	(*═════════════════════════════════════════════════════════*)
	(*  Communication and PLC    *)
	(*═════════════════════════════════════════════════════════*)
	PLC_r_CPUload                                              , (* REAL *)
	PLC_e_ProfinetState                                        , (* eNetcomState *)
	PLC_e_EthercatState                                        , (* eNetcomState *)
	Cooling_CoolingSystemMode                                  , (* eCoolingSystemState *)
	Cooling_HeatPumpStatus                                     , (* eHeatPumpState *)
	Cooling_r_CoolantTemperature                               , (* REAL *)
	Cooling_r_CoolantPressure                                  , (* REAL *)
	Cooling_r_EnclosureDewpoint                                , (* REAL *)
	Cooling_ui_DehumRemainingTime                              , (* UINT *)
	Cooling_HeatPumpSystem_HeatPumpStatus                      , (* eHeatPumpState *)
	Cooling_HeatPumpSystem_PrimaryHeatpumpGet_HeatPumpState    , (* eHeatPumpState *)
	Cooling_HeatPumpSystem_PrimaryHeatpumpGet_Setpoint         , (* REAL *)
	Cooling_HeatPumpSystem_PrimaryHeatpumpGet_Events_b_CommWarning, (* BOOL *)
	Cooling_HeatPumpSystem_PrimaryHeatpumpGet_Events_b_ProbeError, (* BOOL *)
	Cooling_HeatPumpSystem_PrimaryHeatpumpGet_Events_b_PressureError, (* BOOL *)
	Cooling_HeatPumpSystem_PrimaryHeatpumpGet_Events_b_CompressorError, (* BOOL *)
	Cooling_HeatPumpSystem_PrimaryHeatpumpGet_Events_b_ValveError, (* BOOL *)
	Cooling_HeatPumpSystem_PrimaryHeatpumpGet_Events_b_FanError, (* BOOL *)
	Cooling_HeatPumpSystem_PrimaryHeatpumpGet_Events_b_PumpError, (* BOOL *)
	Cooling_HeatPumpSystem_PrimaryHeatpumpGet_Events_b_WaterTempError, (* BOOL *)
	Cooling_HeatPumpSystem_PrimaryHeatpumpGet_Events_b_IOError , (* BOOL *)
	Cooling_HeatPumpSystem_PrimaryHeatpumpGet_Events_b_HeatpumpPreheatingActive, (* BOOL *)
	Cooling_HeatPumpSystem_PrimaryHeatpumpGet_Events_b_TooColdForHeatpumpHeating, (* BOOL *)
	Cooling_HeatPumpSystem_PrimaryHeatpumpGet_HeatpumpData_i_FW_Version, (* INT *)
	Cooling_HeatPumpSystem_PrimaryHeatpumpGet_HeatpumpData_i_FW_release, (* INT *)
	Cooling_HeatPumpSystem_PrimaryHeatpumpGet_HeatpumpData_w_FW_Subrelease, (* WORD *)
	Cooling_HeatPumpSystem_PrimaryHeatpumpGet_HeatpumpData_w_FW_creationDate, (* WORD *)
	Cooling_HeatPumpSystem_PrimaryHeatpumpGet_HeatpumpData_w_Serialnumber_0  , (* WORD *)
	Cooling_HeatPumpSystem_PrimaryHeatpumpGet_HeatpumpData_w_Serialnumber_1  , (* WORD *)
	Cooling_HeatPumpSystem_PrimaryHeatpumpGet_HeatpumpData_w_Serialnumber_2  , (* WORD *)
	Cooling_HeatPumpSystem_PrimaryHeatpumpGet_HeatpumpData_w_Serialnumber_3  , (* WORD *)
	Cooling_HeatPumpSystem_PrimaryHeatpumpGet_HeatpumpData_w_Serialnumber_4  , (* WORD *)
	Cooling_HeatPumpSystem_PrimaryHeatpumpGet_HeatpumpData_w_Serialnumber_5  , (* WORD *)
	Cooling_HeatPumpSystem_PrimaryHeatpumpGet_HeatpumpData_w_Serialnumber_6  , (* WORD *)
	Cooling_HeatPumpSystem_PrimaryHeatpumpGet_HeatpumpData_w_Serialnumber_7  , (* WORD *)
	Cooling_HeatPumpSystem_PrimaryHeatpumpGet_HeatpumpData_w_Serialnumber_8  , (* WORD *)
	Cooling_HeatPumpSystem_PrimaryHeatpumpGet_HeatpumpData_w_Serialnumber_9  , (* WORD *)
	Cooling_HeatPumpSystem_PrimaryHeatpumpGet_HeatpumpData_w_Serialnumber_10 , (* WORD *)
	Cooling_HeatPumpSystem_PrimaryHeatpumpGet_HeatpumpData_w_Serialnumber_11 , (* WORD *)
	Cooling_HeatPumpSystem_PrimaryHeatpumpGet_HeatpumpData_w_Serialnumber_12 , (* WORD *)
	Cooling_HeatPumpSystem_PrimaryHeatpumpGet_HeatpumpData_w_Serialnumber_13 , (* WORD *)
	Cooling_HeatPumpSystem_PrimaryHeatpumpGet_HeatpumpData_w_Serialnumber_14 , (* WORD *)
	Cooling_HeatPumpSystem_PrimaryHeatpumpGet_HeatpumpData_w_Serialnumber_15 , (* WORD *)
	Cooling_HeatPumpSystem_PrimaryHeatpumpGet_HeatpumpData_w_Serialnumber_16 , (* WORD *)
	Cooling_HeatPumpSystem_PrimaryHeatpumpGet_HeatpumpData_w_Serialnumber_17 , (* WORD *)
	Cooling_HeatPumpSystem_PrimaryHeatpumpGet_HeatpumpData_i_OperatingHours, (* INT *)
	Cooling_HeatPumpSystem_PrimaryHeatpumpGet_HeatpumpData_r_CoolantPower, (* REAL *)
	Cooling_HeatPumpSystem_PrimaryHeatpumpGet_HeatpumpData_r_InletWaterTemp, (* REAL *)
	Cooling_HeatPumpSystem_PrimaryHeatpumpGet_HeatpumpData_r_OutletWaterTemp, (* REAL *)
	Cooling_HeatPumpSystem_PrimaryHeatpumpGet_HeatpumpData_r_HighPressure, (* REAL *)
	Cooling_HeatPumpSystem_PrimaryHeatpumpGet_HeatpumpData_r_LowPressure, (* REAL *)
	Cooling_HeatPumpSystem_PrimaryHeatpumpGet_HeatpumpData_r_CompInputTemp, (* REAL *)
	Cooling_HeatPumpSystem_PrimaryHeatpumpGet_HeatpumpData_r_OutdoorTemp, (* REAL *)
	Cooling_HeatPumpSystem_PrimaryHeatpumpGet_HeatpumpData_r_CompOutputTemp, (* REAL *)
	Cooling_HeatPumpSystem_PrimaryHeatpumpGet_HeatpumpData_ui_WaterFlowRate, (* UINT *)
	Cooling_HeatPumpSystem_PrimaryHeatpumpGet_HeatpumpData_w_ErrorList_1  , (* WORD *)
	Cooling_HeatPumpSystem_PrimaryHeatpumpGet_HeatpumpData_w_ErrorList_2  , (* WORD *)
	Cooling_HeatPumpSystem_PrimaryHeatpumpGet_HeatpumpData_w_ErrorList_3  , (* WORD *)
	Cooling_HeatPumpSystem_PrimaryHeatpumpGet_HeatpumpData_w_ErrorList_4  , (* WORD *)
	Cooling_HeatPumpSystem_PrimaryHeatpumpGet_HeatpumpData_w_ErrorList_5  , (* WORD *)
	Cooling_HeatPumpSystem_PrimaryHeatpumpGet_HeatpumpData_w_ErrorList_6  , (* WORD *)
	Cooling_HeatPumpSystem_PrimaryHeatpumpGet_HeatpumpData_w_ErrorList_7  , (* WORD *)
	Cooling_HeatPumpSystem_PrimaryHeatpumpGet_HeatpumpData_r_FanSpeedPCT, (* REAL *)
	Cooling_HeatPumpSystem_PrimaryHeatpumpGet_HeatpumpData_r_PumpSpeedPCT, (* REAL *)
	Cooling_HeatPumpSystem_PrimaryHeatpumpGet_HeatpumpData_r_SetpointHeating, (* REAL *)
	Cooling_HeatPumpSystem_PrimaryHeatpumpGet_HeatpumpData_r_SetpointCooling, (* REAL *)
	Cooling_HeatPumpSystem_PrimaryHeatpumpGet_HeatpumpData_b_DefrostingActive, (* BOOL *)
	Cooling_HeatPumpSystem_SecondaryHeatpumpGet_HeatPumpState  , (* eHeatPumpState *)
	Cooling_HeatPumpSystem_SecondaryHeatpumpGet_Setpoint       , (* REAL *)
	Cooling_HeatPumpSystem_SecondaryHeatpumpGet_Events_b_CommWarning, (* BOOL *)
	Cooling_HeatPumpSystem_SecondaryHeatpumpGet_Events_b_ProbeError, (* BOOL *)
	Cooling_HeatPumpSystem_SecondaryHeatpumpGet_Events_b_PressureError, (* BOOL *)
	Cooling_HeatPumpSystem_SecondaryHeatpumpGet_Events_b_CompressorError, (* BOOL *)
	Cooling_HeatPumpSystem_SecondaryHeatpumpGet_Events_b_ValveError, (* BOOL *)
	Cooling_HeatPumpSystem_SecondaryHeatpumpGet_Events_b_FanError, (* BOOL *)
	Cooling_HeatPumpSystem_SecondaryHeatpumpGet_Events_b_PumpError, (* BOOL *)
	Cooling_HeatPumpSystem_SecondaryHeatpumpGet_Events_b_WaterTempError, (* BOOL *)
	Cooling_HeatPumpSystem_SecondaryHeatpumpGet_Events_b_IOError, (* BOOL *)
	Cooling_HeatPumpSystem_SecondaryHeatpumpGet_Events_b_HeatpumpPreheatingActive, (* BOOL *)
	Cooling_HeatPumpSystem_SecondaryHeatpumpGet_Events_b_TooColdForHeatpumpHeating, (* BOOL *)
	Cooling_HeatPumpSystem_SecondaryHeatpumpGet_HeatpumpData_i_FW_Version, (* INT *)
	Cooling_HeatPumpSystem_SecondaryHeatpumpGet_HeatpumpData_i_FW_release, (* INT *)
	Cooling_HeatPumpSystem_SecondaryHeatpumpGet_HeatpumpData_w_FW_Subrelease, (* WORD *)
	Cooling_HeatPumpSystem_SecondaryHeatpumpGet_HeatpumpData_w_FW_creationDate, (* WORD *)
	Cooling_HeatPumpSystem_SecondaryHeatpumpGet_HeatpumpData_w_Serialnumber_0  , (* WORD *)
	Cooling_HeatPumpSystem_SecondaryHeatpumpGet_HeatpumpData_w_Serialnumber_1  , (* WORD *)
	Cooling_HeatPumpSystem_SecondaryHeatpumpGet_HeatpumpData_w_Serialnumber_2  , (* WORD *)
	Cooling_HeatPumpSystem_SecondaryHeatpumpGet_HeatpumpData_w_Serialnumber_3  , (* WORD *)
	Cooling_HeatPumpSystem_SecondaryHeatpumpGet_HeatpumpData_w_Serialnumber_4  , (* WORD *)
	Cooling_HeatPumpSystem_SecondaryHeatpumpGet_HeatpumpData_w_Serialnumber_5  , (* WORD *)
	Cooling_HeatPumpSystem_SecondaryHeatpumpGet_HeatpumpData_w_Serialnumber_6  , (* WORD *)
	Cooling_HeatPumpSystem_SecondaryHeatpumpGet_HeatpumpData_w_Serialnumber_7  , (* WORD *)
	Cooling_HeatPumpSystem_SecondaryHeatpumpGet_HeatpumpData_w_Serialnumber_8  , (* WORD *)
	Cooling_HeatPumpSystem_SecondaryHeatpumpGet_HeatpumpData_w_Serialnumber_9  , (* WORD *)
	Cooling_HeatPumpSystem_SecondaryHeatpumpGet_HeatpumpData_w_Serialnumber_10 , (* WORD *)
	Cooling_HeatPumpSystem_SecondaryHeatpumpGet_HeatpumpData_w_Serialnumber_11 , (* WORD *)
	Cooling_HeatPumpSystem_SecondaryHeatpumpGet_HeatpumpData_w_Serialnumber_12 , (* WORD *)
	Cooling_HeatPumpSystem_SecondaryHeatpumpGet_HeatpumpData_w_Serialnumber_13 , (* WORD *)
	Cooling_HeatPumpSystem_SecondaryHeatpumpGet_HeatpumpData_w_Serialnumber_14 , (* WORD *)
	Cooling_HeatPumpSystem_SecondaryHeatpumpGet_HeatpumpData_w_Serialnumber_15 , (* WORD *)
	Cooling_HeatPumpSystem_SecondaryHeatpumpGet_HeatpumpData_w_Serialnumber_16 , (* WORD *)
	Cooling_HeatPumpSystem_SecondaryHeatpumpGet_HeatpumpData_w_Serialnumber_17 , (* WORD *)
	Cooling_HeatPumpSystem_SecondaryHeatpumpGet_HeatpumpData_i_OperatingHours, (* INT *)
	Cooling_HeatPumpSystem_SecondaryHeatpumpGet_HeatpumpData_r_CoolantPower, (* REAL *)
	Cooling_HeatPumpSystem_SecondaryHeatpumpGet_HeatpumpData_r_InletWaterTemp, (* REAL *)
	Cooling_HeatPumpSystem_SecondaryHeatpumpGet_HeatpumpData_r_OutletWaterTemp, (* REAL *)
	Cooling_HeatPumpSystem_SecondaryHeatpumpGet_HeatpumpData_r_HighPressure, (* REAL *)
	Cooling_HeatPumpSystem_SecondaryHeatpumpGet_HeatpumpData_r_LowPressure, (* REAL *)
	Cooling_HeatPumpSystem_SecondaryHeatpumpGet_HeatpumpData_r_CompInputTemp, (* REAL *)
	Cooling_HeatPumpSystem_SecondaryHeatpumpGet_HeatpumpData_r_OutdoorTemp, (* REAL *)
	Cooling_HeatPumpSystem_SecondaryHeatpumpGet_HeatpumpData_r_CompOutputTemp, (* REAL *)
	Cooling_HeatPumpSystem_SecondaryHeatpumpGet_HeatpumpData_ui_WaterFlowRate, (* UINT *)
	Cooling_HeatPumpSystem_SecondaryHeatpumpGet_HeatpumpData_w_ErrorList_1  , (* WORD *)
	Cooling_HeatPumpSystem_SecondaryHeatpumpGet_HeatpumpData_w_ErrorList_2  , (* WORD *)
	Cooling_HeatPumpSystem_SecondaryHeatpumpGet_HeatpumpData_w_ErrorList_3  , (* WORD *)
	Cooling_HeatPumpSystem_SecondaryHeatpumpGet_HeatpumpData_w_ErrorList_4  , (* WORD *)
	Cooling_HeatPumpSystem_SecondaryHeatpumpGet_HeatpumpData_w_ErrorList_5  , (* WORD *)
	Cooling_HeatPumpSystem_SecondaryHeatpumpGet_HeatpumpData_w_ErrorList_6  , (* WORD *)
	Cooling_HeatPumpSystem_SecondaryHeatpumpGet_HeatpumpData_w_ErrorList_7  , (* WORD *)
	Cooling_HeatPumpSystem_SecondaryHeatpumpGet_HeatpumpData_r_FanSpeedPCT, (* REAL *)
	Cooling_HeatPumpSystem_SecondaryHeatpumpGet_HeatpumpData_r_PumpSpeedPCT, (* REAL *)
	Cooling_HeatPumpSystem_SecondaryHeatpumpGet_HeatpumpData_r_SetpointHeating, (* REAL *)
	Cooling_HeatPumpSystem_SecondaryHeatpumpGet_HeatpumpData_r_SetpointCooling, (* REAL *)
	Cooling_HeatPumpSystem_SecondaryHeatpumpGet_HeatpumpData_b_DefrostingActive, (* BOOL *)
	Cooling_Events_b_SystemOvertemperatureWarning              , (* BOOL *)
	Cooling_Events_b_SystemUnderTemperatureWarning             , (* BOOL *)
	Cooling_Events_b_CoolingSystemFuseFailure                  , (* BOOL *)
	Cooling_Events_b_ACwaterPumpTimeOut                        , (* BOOL *)
	Cooling_Events_b_InverterLoopValveStuck                    , (* BOOL *)
	Cooling_Events_b_BattLoopValveStuck                        , (* BOOL *)
	Cooling_Events_b_FancoilLoopValveStuck                     , (* BOOL *)
	Cooling_Events_b_DCpumpPressureFault                       , (* BOOL *)
	Cooling_Events_b_DCpumpTimeout                             , (* BOOL *)
	Cooling_Events_b_CoolingLoopIdlePressureWarning            , (* BOOL *)
	Cooling_Events_b_CoolingLoopIdlePressureError              , (* BOOL *)
	Cooling_Events_b_InverterCoolingLoopError                  , (* BOOL *)
	Cooling_Events_b_HeatpumpWarning                           , (* BOOL *)
	Cooling_Events_b_HeatPumpError                             , (* BOOL *)
	Cooling_Events_b_CoolantTempTooLow                         , (* BOOL *)
	Cooling_Events_b_CoolantTempLow                            , (* BOOL *)
	Cooling_Events_b_CoolantTempTooHigh                        , (* BOOL *)
	Cooling_Events_b_CoolantTempHigh                           , (* BOOL *)
	Router_Device_SystemUptime                                 , (* UDINT *)
	Router_Device_Temperature                                  , (* REAL *)
	Router_Device_RouterSerial                                 , (* STRING(32) *)
	Router_GPS_Latitude                                        , (* REAL *)
	Router_GPS_Longitude                                       , (* REAL *)
	Router_GPS_FixTime                                         , (* STRING(32) *)
	Router_GPS_DateTime                                        , (* DT *)
	Router_GPS_Speed                                           , (* REAL *)
	Router_GPS_SatCount                                        , (* UINT *)
	Router_GPS_Accuracy                                        , (* REAL *)
	Router_Mobile_NetworkOperator                              , (* STRING(32) *)
	Router_Mobile_NetworkInfo                                  , (* STRING(32) *)
	Router_Mobile_NetworkType                                  , (* STRING(32) *)
	Router_Mobile_RSSI                                         , (* DINT *)
	Router_Mobile_ui_Sim1DataSendMonth                         , (* UINT *)
	Router_Mobile_ui_Sim1DataReceivedMonth                     , (* UINT *)
	Router_Mobile_ui_Sim2DataSendMonth                         , (* UINT *)
	Router_Mobile_ui_Sim2DataReceivedMonth                     , (* UINT *)
	Router_Mobile_s_EmergencySMSNumber                         , (* STRING(20) *)
	Router_Mobile_s_SecondarySMSNumber                         , (* STRING(20) *)
	Router_Mobile_s_EmergencySMSDevName                        , (* STRING(18) *)
	Router_Mobile_st_LatestSMSMessage                          , (* STRING(80) *)
	Router_Mobile_ModemState                                   , (* eModemState *)
	Router_Mobile_NetworkState                                 , (* eNetworkState *)
	Router_Mobile_ui_ActiveSim                                 , (* UINT *)
	Router_Mobile_SimStatus                                    , (* eSimState *)
	Router_Wifi_WifiClienModeStatus                            , (* eWifiStatus *)
	Router_Wifi_WifiAPModeStatus                               , (* eWifiStatus *)
	Router_Wifi_WifiApNumberOfClients                          , (* UINT *)
	Router_e_SMSStatus                                         , (* eSMSStatus *)
	Router_Events_b_MBCommWarning                              , (* BOOL *)
	Router_Events_b_NoSimWarning                               , (* BOOL *)
	Router_Events_b_NoNetworkWarning                           , (* BOOL *)
	Router_Events_b_noGPSFixWarning                            , (* BOOL *)
	Router_Events_b_SMSNotSendError                            , (* BOOL *)
	Router_Events_b_NoSMSNumberAvailable                       , (* BOOL *)
	Router_Events_b_TimeUpdateFailed                           , (* BOOL *)

	(*═════════════════════════════════════════════════════════*)
	(*  External Systems and I/O    *)
	(*═════════════════════════════════════════════════════════*)
	controlfb_control_b_start                                  , (* BOOL *)
	controlfb_control_b_stop                                   , (* BOOL *)
	controlfb_control_b_shutdown                               , (* BOOL *)
	controlfb_control_b_Reset                                  , (* BOOL *)
	controlfb_control_b_SystemShutdown                         , (* BOOL *)
	controlfb_control_b_EMstop                                 , (* BOOL *)
	controlfb_control_b_ClearHistory                           , (* BOOL *)
	controlfb_control_b_ActivateSettings                       , (* BOOL *)
	controlfb_control_b_startDeHum                             , (* BOOL *)
	controlfb_Operation_inputgrid_b_SyncClose                  , (* BOOL *)
	controlfb_Operation_Genset_b_manualStart                   , (* BOOL *)
	controlfb_Operation_PSB_b_SyncClose                        , (* BOOL *)
	controlfb_Operation_charger_b_StartCharging                , (* BOOL *)
	controlfb_Operation_charger_b_ResetCharger                 , (* BOOL *)
	controlfb_Operation_system_r_NominalVoltage                , (* REAL *)
	controlfb_Operation_system_r_NominalFrequency              , (* REAL *)
	controlfb_Operation_system_r_Pset                          , (* REAL *)
	controlfb_Operation_system_r_Qset                          , (* REAL *)
	controlfb_Operation_system_r_PFset                         , (* REAL *)
	controlfb_Operation_system_b_PFsetEnable                   , (* BOOL *)
	controlfb_Operation_system_b_SounderMute                   , (* BOOL *)
	controlfb_Operation_system_b_SounderTest                   , (* BOOL *)
	controlfb_Operation_system_b_GenGridModeTrans              , (* BOOL *)
	controlfb_Operation_system_b_GridTakeOverEnable            , (* BOOL *)
	controlfb_Operation_parallel_b_DetectSlaves                , (* BOOL *)
	controlfb_Operation_parallel_r_ActivePowerSlave1           , (* REAL *)
	controlfb_Operation_parallel_r_ReactivePowerSlave1         , (* REAL *)
	controlfb_Operation_parallel_r_ActivePowerSlave2           , (* REAL *)
	controlfb_Operation_parallel_r_ReactivePowerSlave2         , (* REAL *)
	controlfb_Operation_BMS_b_ManualStartHVDC                  , (* BOOL *)
	controlfb_SoftSettings_inputgrid_PeakshaveMode             , (* ePeakshaveMode *)
	controlfb_SoftSettings_inputgrid_setpointTimeslot1_r_SocTarget, (* REAL *)
	controlfb_SoftSettings_inputgrid_setpointTimeslot1_r_IdleChargePower, (* REAL *)
	controlfb_SoftSettings_inputgrid_setpointTimeslot1_r_FeedInCurrentLimitSoft, (* REAL *)
	controlfb_SoftSettings_inputgrid_setpointTimeslot1_r_SupplyCurrentLimitSoft, (* REAL *)
	controlfb_SoftSettings_inputgrid_setpointTimeslot2_r_SocTarget, (* REAL *)
	controlfb_SoftSettings_inputgrid_setpointTimeslot2_r_IdleChargePower, (* REAL *)
	controlfb_SoftSettings_inputgrid_setpointTimeslot2_r_FeedInCurrentLimitSoft, (* REAL *)
	controlfb_SoftSettings_inputgrid_setpointTimeslot2_r_SupplyCurrentLimitSoft, (* REAL *)
	controlfb_SoftSettings_inputgrid_b_BreakerControl          , (* BOOL *)
	controlfb_SoftSettings_inputgrid_b_ReverseCTDirection      , (* BOOL *)
	controlfb_SoftSettings_inputgrid_ui_CTrange                , (* UINT *)
	controlfb_SoftSettings_inputgrid_r_VTratio                 , (* REAL *)
	controlfb_SoftSettings_inputgrid_b_GridCodesActive         , (* BOOL *)
	controlfb_SoftSettings_inputgrid_b_WeakGridInput           , (* BOOL *)
	controlfb_SoftSettings_inputgrid_breaker_AutoConnect       , (* BOOL *)
	controlfb_SoftSettings_inputgrid_breaker_ShutdownDisconnect, (* BOOL *)
	controlfb_SoftSettings_inputgrid_breaker_EMstopDisconnect  , (* BOOL *)
	controlfb_SoftSettings_inputgrid_breaker_CurrentLimitDisconnect, (* BOOL *)
	controlfb_SoftSettings_inputgrid_breaker_CurrentLimitRetries, (* BYTE *)
	controlfb_SoftSettings_inputgenset_b_AutoStartStop         , (* BOOL *)
	controlfb_SoftSettings_inputgenset_b_HydridMode            , (* BOOL *)
	controlfb_SoftSettings_inputgenset_b_EnableSchedule        , (* BOOL *)
	controlfb_SoftSettings_inputgenset_setpointTimeslot1_r_SoCStart, (* REAL *)
	controlfb_SoftSettings_inputgenset_setpointTimeslot1_r_SoCStop, (* REAL *)
	controlfb_SoftSettings_inputgenset_setpointTimeslot1_r_BatteryloadStart, (* REAL *)
	controlfb_SoftSettings_inputgenset_setpointTimeslot1_r_BatteryloadStop, (* REAL *)
	controlfb_SoftSettings_inputgenset_setpointTimeslot1_b_StartAtBatteryError, (* BOOL *)
	controlfb_SoftSettings_inputgenset_setpointTimeslot2_r_SoCStart, (* REAL *)
	controlfb_SoftSettings_inputgenset_setpointTimeslot2_r_SoCStop, (* REAL *)
	controlfb_SoftSettings_inputgenset_setpointTimeslot2_r_BatteryloadStart, (* REAL *)
	controlfb_SoftSettings_inputgenset_setpointTimeslot2_r_BatteryloadStop, (* REAL *)
	controlfb_SoftSettings_inputgenset_setpointTimeslot2_b_StartAtBatteryError, (* BOOL *)
	controlfb_SoftSettings_inputgenset_b_PSBExtGensetMonitoring, (* BOOL *)
	controlfb_SoftSettings_inputgenset_b_FreqProtectionEnable  , (* BOOL *)
	controlfb_SoftSettings_inputgenset_Generator_e_GensetMode  , (* eGensetMode *)
	controlfb_SoftSettings_inputgenset_Generator_b_GensetLoadshareLine, (* BOOL *)
	controlfb_SoftSettings_inputgenset_Generator_r_RatedPower  , (* REAL *)
	controlfb_SoftSettings_inputgenset_Generator_r_powerloadMax, (* REAL *)
	controlfb_SoftSettings_inputgenset_Generator_r_PowerloadMin, (* REAL *)
	controlfb_SoftSettings_inputgenset_Generator_r_PowerloadEff, (* REAL *)
	controlfb_SoftSettings_inputgenset_Generator_r_ramprate    , (* REAL *)
	controlfb_SoftSettings_inputgenset_Generator_ui_CooldownTime, (* UINT *)
	controlfb_SoftSettings_inputgenset_Generator_ui_WarmupTime , (* UINT *)
	controlfb_SoftSettings_inputgenset_Loadbank_b_Enable       , (* BOOL *)
	controlfb_SoftSettings_inputgenset_Loadbank_r_PowerRating  , (* REAL *)
	controlfb_SoftSettings_inputgenset_Loadbank_r_PowerStepSize, (* REAL *)
	controlfb_SoftSettings_PSB_PeakshaveMode                   , (* ePeakshaveMode *)
	controlfb_SoftSettings_PSB_setpointTimeslot1_r_SocTarget   , (* REAL *)
	controlfb_SoftSettings_PSB_setpointTimeslot1_r_IdleChargePower, (* REAL *)
	controlfb_SoftSettings_PSB_setpointTimeslot1_r_FeedInCurrentLimitSoft, (* REAL *)
	controlfb_SoftSettings_PSB_setpointTimeslot1_r_SupplyCurrentLimitSoft, (* REAL *)
	controlfb_SoftSettings_PSB_setpointTimeslot2_r_SocTarget   , (* REAL *)
	controlfb_SoftSettings_PSB_setpointTimeslot2_r_IdleChargePower, (* REAL *)
	controlfb_SoftSettings_PSB_setpointTimeslot2_r_FeedInCurrentLimitSoft, (* REAL *)
	controlfb_SoftSettings_PSB_setpointTimeslot2_r_SupplyCurrentLimitSoft, (* REAL *)
	controlfb_SoftSettings_PSB_b_BreakerControl                , (* BOOL *)
	controlfb_SoftSettings_PSB_b_ReverseCTDirection            , (* BOOL *)
	controlfb_SoftSettings_PSB_ui_CTrange                      , (* UINT *)
	controlfb_SoftSettings_PSB_r_VTratio                       , (* REAL *)
	controlfb_SoftSettings_system_b_EnableSchedule             , (* BOOL *)
	controlfb_SoftSettings_system_b_EnableTransportMode        , (* BOOL *)
	controlfb_SoftSettings_system_b_EcoModeEnable              , (* BOOL *)
	controlfb_SoftSettings_system_e_UgridPowerMode             , (* eUgridPowerMode *)
	controlfb_SoftSettings_system_e_NetcontactorMode           , (* eNetcontMode *)
	controlfb_SoftSettings_system_e_UgridPowerLimitingMode     , (* ePLM *)
	controlfb_SoftSettings_system_b_AutomaticSwitching         , (* BOOL *)
	controlfb_SoftSettings_system_b_AMF                        , (* BOOL *)
	controlfb_SoftSettings_system_r_FrequencyDroop             , (* REAL *)
	controlfb_SoftSettings_system_r_VoltageDroop               , (* REAL *)
	controlfb_SoftSettings_system_r_SocMin                     , (* REAL *)
	controlfb_SoftSettings_system_r_SocMax                     , (* REAL *)
	controlfb_SoftSettings_system_r_PDischargeLimit            , (* REAL *)
	controlfb_SoftSettings_system_r_PChargeLimit               , (* REAL *)
	controlfb_SoftSettings_system_r_AMax                       , (* REAL *)
	controlfb_SoftSettings_system_s_SystemName                 , (* STRING(18) *)
	controlfb_SoftSettings_system_s_SMSnumber                  , (* STRING(18) *)
	controlfb_SoftSettings_system_ScheduleTimeSlot1_b_active   , (* BOOL *)
	controlfb_SoftSettings_system_ScheduleTimeSlot1_usi_DayOfWeek, (* USINT *)
	controlfb_SoftSettings_system_ScheduleTimeSlot1_usi_HourOfDay, (* USINT *)
	controlfb_SoftSettings_system_ScheduleTimeSlot1_usi_MinuteOfHour, (* USINT *)
	controlfb_SoftSettings_system_ScheduleTimeSlot2_b_active   , (* BOOL *)
	controlfb_SoftSettings_system_ScheduleTimeSlot2_usi_DayOfWeek, (* USINT *)
	controlfb_SoftSettings_system_ScheduleTimeSlot2_usi_HourOfDay, (* USINT *)
	controlfb_SoftSettings_system_ScheduleTimeSlot2_usi_MinuteOfHour, (* USINT *)
	controlfb_SoftSettings_system_by_LEDbrightness             , (* BYTE *)
	controlfb_SoftSettings_setup_e_AcInputType                 , (* eAcInputType *)
	controlfb_SoftSettings_setup_b_MasterSlaveMode             , (* BOOL *)
	controlfb_SoftSettings_setup_b_PeakshaveBoxEnable          , (* BOOL *)
	controlfb_SoftSettings_setup_e_Gridmode                    , (* eGridmode *)
	controlfb_SoftSettings_setup_e_DcCouplingType              , (* eDCinputType *)
	controlfb_SoftSettings_setup_b_ExtGenset                   , (* BOOL *)
	controlfb_HardSettings_setup_e_ControlSource               , (* eControlSources *)
	controlfb_HardSettings_charger_r_PowerMax                  , (* REAL *)
	controlfb_HardSettings_parallel_b_MasterSlaveEnabled       , (* BOOL *)
	controlfb_HardSettings_parallel_b_UnitIsMaster             , (* BOOL *)
	controlfb_HardSettings_parallel_b_ShutdownOnCommError      , (* BOOL *)
	controlfb_HardSettings_parallel_b_EffiencyMode             , (* BOOL *)
	controlfb_HardSettings_parallel_r_VoltageDroop             , (* REAL *)
	controlfb_HardSettings_parallel_r_FrequencyDroop           , (* REAL *)
	controlfb_HardSettings_system_r_PDischargeLimit            , (* REAL *)
	controlfb_HardSettings_system_r_PChargeLimit               , (* REAL *)
	controlfb_HardSettings_system_r_SMax                       , (* REAL *)
	controlfb_HardSettings_system_r_Amax                       , (* REAL *)
	controlfb_HardSettings_system_e_EarthingSystem             , (* eEarthingSystems *)
	controlfb_HardSettings_system_a_ui_InputCurrentLimit_1     , (* UINT *)
	controlfb_HardSettings_system_a_ui_InputCurrentLimit_2     , (* UINT *)
	controlfb_HardSettings_system_a_ui_OutputCurrentLimit_1    , (* UINT *)
	controlfb_HardSettings_system_a_ui_OutputCurrentLimit_2    , (* UINT *)
	controlfb_HardSettings_system_a_ui_OutputCurrentLimit_3    , (* UINT *)
	Generator_CommunicationOK                                  , (* BOOL *)
	Generator_FuelLow                                          , (* BOOL *)
	Generator_FuelCritical                                     , (* BOOL *)
	Generator_bGenBreakerClosed                                , (* BOOL *)
	Generator_bMainBreakerClosed                               , (* BOOL *)
	Generator_bGenRunning                                      , (* BOOL *)
	Generator_bGenVoltFreqOK                                   , (* BOOL *)
	Generator_bMainsFailure                                    , (* BOOL *)
	Generator_eActiveGenMode                                   , (* eGenOperationMode *)
	Generator_bIslandModeActive                                , (* BOOL *)
	Generator_bAMFActive                                       , (* BOOL *)
	Generator_bPeakshaveActive                                 , (* BOOL *)
	Generator_bFixedPowerActive                                , (* BOOL *)
	Generator_ar_LineVoltage_AVG                               , (* REAL *)
	Generator_ar_LineVoltage_L1                                , (* REAL *)
	Generator_ar_LineVoltage_L2                                , (* REAL *)
	Generator_ar_LineVoltage_L3                                , (* REAL *)
	Generator_ar_PhaseVoltage_AVG                              , (* REAL *)
	Generator_ar_PhaseVoltage_L1                               , (* REAL *)
	Generator_ar_PhaseVoltage_L2                               , (* REAL *)
	Generator_ar_PhaseVoltage_L3                               , (* REAL *)
	Generator_ar_Frequency_AVG                                 , (* REAL *)
	Generator_ar_Frequency_L1                                  , (* REAL *)
	Generator_ar_Frequency_L2                                  , (* REAL *)
	Generator_ar_Frequency_L3                                  , (* REAL *)
	Generator_ar_Current_AVG                                   , (* REAL *)
	Generator_ar_Current_L1                                    , (* REAL *)
	Generator_ar_Current_L2                                    , (* REAL *)
	Generator_ar_Current_L3                                    , (* REAL *)
	Generator_ar_PowerFactor_AVG                               , (* REAL *)
	Generator_ar_ActivePower_AVG                               , (* REAL *)
	Generator_ar_ActivePower_L1                                , (* REAL *)
	Generator_ar_ActivePower_L2                                , (* REAL *)
	Generator_ar_ActivePower_L3                                , (* REAL *)
	Generator_ar_ReactivePower_AVG                             , (* REAL *)
	Generator_ar_ApparentPower_AVG                             , (* REAL *)
	HartingIO_b_DigitalInput1Active                            , (* BOOL *)
	HartingIO_b_DigitalInput2Active                            , (* BOOL *)
	HartingIO_b_GenLowFuel                                     , (* BOOL *)
	HartingIO_b_ExtSystemShutdownRequest                       , (* BOOL *)
	HartingIO_b_ExtEMstopOK                                    , (* BOOL *)
	HartingIO_b_ExtEMstopActive                                , (* BOOL *)
	last
) DINT;
END_TYPE

(* stored: Version 1.1.0.1, ProductVersion 3.1.4026.18
   DUT eDataMappingVarNames: Id {5ee32b74-8fd4-4bb0-b3f8-4847515968ac} *)
